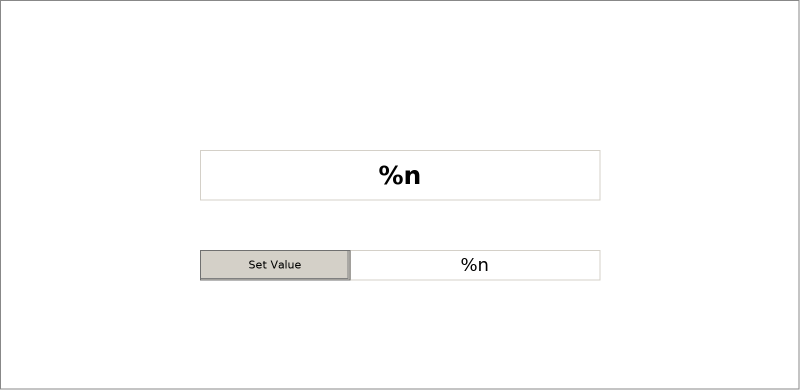
VISUALIZATION VisuKL15XXControl  // 800x390
VAR_IN_OUT
	fbManualControler	: FB_ManualController ;
END_VAR
    Textfield (200,150 400x50), "%n", text variable: fbManualControler.pDevKL1512^.stManualControl.nCount
    Textfield (350,250 250x30), "%n", text variable: fbManualControler.pDevKL1512^.stManualControl.nManValue
        OnMouseClick: write the text variable via VisuDialogs.Numpad
    Button (200,250 150x30), "Set Value"
        tap fbManualControler.pDevKL1512^.stManualControl.bManSetValue
END_VISUALIZATION

(* stored: Version 1.1.0.1, ProductVersion 3.1.4024.10
   Visu VisuKL15XXControl: Id {8271f1d5-0bdb-4509-8f23-418c2078db19} *)
